PROGRAM executevolt
VAR
END_VAR

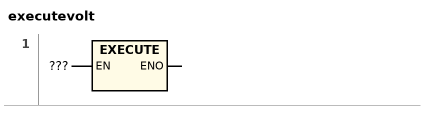
// NETWORK 1

END_PROGRAM

(* stored: Version 1.1.0.1, ProductVersion 3.1.4024.16
   POU executevolt: Id {652280c4-9dd2-41ce-8d48-ce02a548ffe8}, SpecialFunc None *)
